// TIA Portal V20 export
DATA_BLOCK "FB_Fuel_Stand_DB"   // DB8
// stored: InstanceOfName FB_Fuel_Stand, InstanceOfType FB
"FB_Fuel_Stand"
   // VAR_INPUT
   //    iUnscaledMin : Real;
   //    iUnscaledMax : Real;
   //    iScaledMin : Real;
   //    iOffset : Real;
   //    iUnscaledAktVal : Int;
   //    iQuittieren : Bool;
   //    iImpuls : Bool;
   //    iStoerungUnterdr : Bool;
   //    iPipe_diameter : Bool;
   //    iMaxFlowRate : Real;
   //    iTemp_Raw : Word;
   //    Temp_Min : Real;
   //    Temp_Max : Real;
   //    Refrence_Temp : Real;
   //    iAssembly_Place : String;
   // END_VAR
   // VAR_OUTPUT
   //    outputfehler : "UDT_Flowmeter_Stoe";
   // END_VAR
   // VAR
   //    sFlowScaledValue : Real;
   //    eingang_80_plc : Bool;
   //    Buffer : Array[1..10] of Real;
   //    Index : DInt;
   //    Sum : Real;
   //    sScaledMax : Real;
   //    i : Int;
   //    sAvg : Real;
   //    bitte_schalte_an : Bool;
   //    sCyclecount : Real;
   //    IEC_Timer_0_Instance { S7_SetPoint := 'True'} : TON_TIME;
   // END_VAR
BEGIN
END_DATA_BLOCK
